{attribute 'GeneratedUsingTerminal: DL-EC1A-0000'}
{attribute addProperty BoxType "DL-EC1A-0000"}
{attribute addProperty Id "Tool_00_ScoreAT %I*DINT4"}
{attribute addProperty CRC "539608926"}
{attribute addProperty Size "4"}
TYPE ID02_Current_Value_2029C75E EXTENDS InputBase_8311D824 :
STRUCT
	{attribute addProperty Name "Tool_00_Score"}
	Tool_00_Score AT %I* : DINT;
END_STRUCT
END_TYPE

(* stored: Version 1.2.0.0, ProductVersion 3.1.4024.12
   DUT ID02_Current_Value_2029C75E: Id {891dd371-7695-0aed-0b17-e8255dbe2014} *)
